PROGRAM MAIN
VAR
			// UPS variables persistentes
	fbUPS: FB_S_UPS_CX81xx;//Instancia de la UPS
	// Entradas
	id0Local   AT %I*: BYTE;
	id0Remoto1 AT %I*: BYTE;
	// Salidas
	od0Local   AT %Q*: BYTE;
	od0Remoto1 AT %Q*: BYTE;
	fbUtilidades: Utilidades;
END_VAR

fbUPS(iPLCPort:= 851,);
Fecha_Hora_PLC();
FuncParoNodoCorteH4Remote1();
FuncParoNodoMultidiscos();
Events();
fbUtilidades();

END_PROGRAM

(* stored: Version 1.1.0.1, ProductVersion 3.1.4024.12
   POU MAIN: Id {ed129647-f36b-4013-ad91-896499ac6390}, SpecialFunc None *)
